// Block: TokenChain

DATA_BLOCK TokenChain
VERSION : 0.1
   NON_RETAIN
   VAR
      Data : Array[1..TOKENCHAIN_MAX] of TokenChain_Data;
   END_VAR

BEGIN
   // No initialization required
END_DATA_BLOCK
